Staubli VAL3: default.dtx

mdesc mNomSpeed = {blend=joint, accel=100, vel=100, decel=100, tmax=99999, rmax=99999, leave=50, reach=50}
